Staubli VAL3: onFunctionSel.pgx

public program onFunctionSel(num x_nIndex (dimensions=1), string x_sEvent (dimensions=1), num x_nFunctionKey (dimensions=1))
begin
  //
  // do on Key action
  //
  // x_nIndex = actual index item
  // x_sEvent = actual event item
  //
  switch x_nFunctionKey
    // F1 button
    case 271
    break
    // F2 button
    case 272
    break
    // F3 button
    case 273
    break
    // F4 button
    case 274
    break
    // F5 button
    case 275
    break
    // F6 button
    case 276
    break
    // F7 button
    case 277
    break
    // F8 button
    case 278
    break
  endSwitch
end
